TYPE ST_Xbox_Controller_Rumble :
STRUCT
	// Rumble of left motor (0..100%)
	fLeftMotor 	: REAL;
	// Rumble of right motor (0..100%)
	fRightMotor : REAL;
END_STRUCT
END_TYPE

(* stored: Version 1.1.0.1, ProductVersion 3.1.4024.11
   DUT ST_Xbox_Controller_Rumble: Id {b339dff4-fa4d-487e-9d7c-0d56e52c72e7} *)
